RoboDK station: robot_arm.rdk

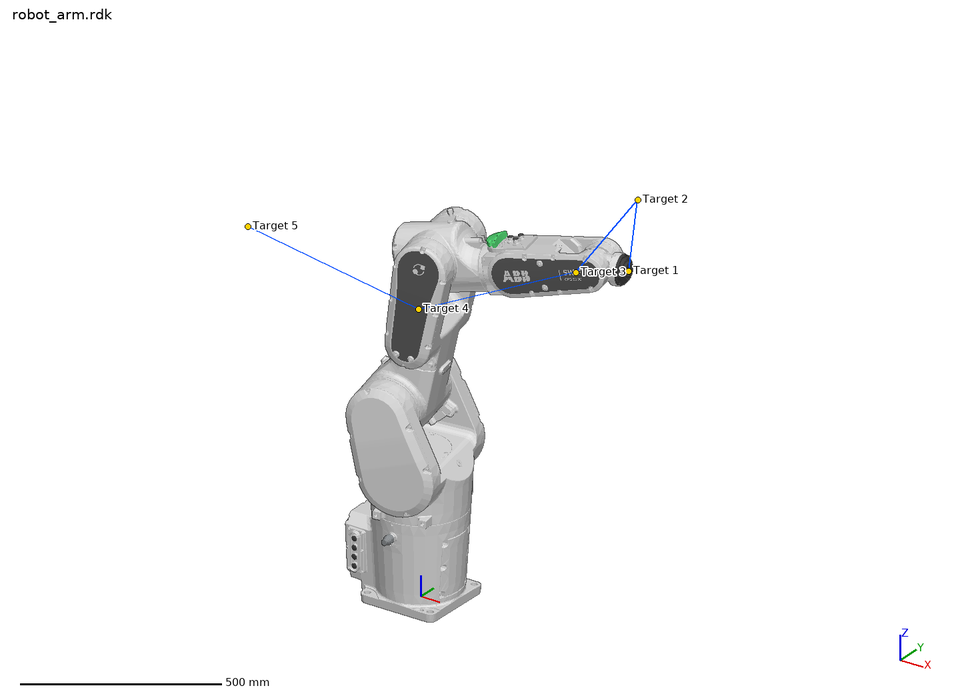
[picture v0: the station drawn from its stored meshes, robots at their saved joint values, targets as dots, program paths as lines]
Station robot_arm (saved by RoboDK 5.8.0). Poses are relative to the parent item; angles as X-Y-Z fixed-axis rotations.
  - frame ABB CRB 1300-11/0.9 Base at (0, 1000, 0) mm
    - robot ABB CRB 1300-11/0.9: 6 axes
        modified DH rows (alpha deg, a mm, theta deg, d mm): 0, 0, 0, 544; -90, 50, -90, 0; 0, 425, 0, 0; -90, 40, 0, 425; 90, 0, 0, 0; -90, 0, 180, 90
        joint limits [-180, -100, -210, -230, -130, -242] to [180, 130, 65, 230, 130, 242]; home [0, 0, 0, 0, 0, 0]; saved at [-169.09, -13.79, -153.79, -179.99, 12.4, 0]
    - target Target 1 (Cartesian target) at (554.75, 106.93, 1009.12) mm, rotated rx 26.03 ry 89.98 rz 36.94 deg; joints [-169.09, -13.79, -153.79, -179.99, 12.4, 0] of ABB CRB 1300-11/0.9
    - target Target 2 (Cartesian target) at (342.12, 449.59, 1009.12) mm, rotated rx 26.03 ry 89.98 rz 78.76 deg; joints [-127.27, -13.79, -153.79, -179.99, 12.4, 0] of ABB CRB 1300-11/0.9
    - target Target 3 (Cartesian target) at (-34.26, 718.46, 596.2) mm, rotated rx 179.98 ry 56.8 rz -87.29 deg; joints [-87.27, -47.01, -153.79, -179.99, 12.4, 0] of ABB CRB 1300-11/0.9
    - target Target 4 (Cartesian target) at (-369.45, 518.9, 480.16) mm, rotated rx 179.98 ry 40.97 rz -54.58 deg; joints [-54.55, -47, -169.64, -179.98, 12.39, 0] of ABB CRB 1300-11/0.9
    - target Target 5 (Cartesian target) at (-573.83, 73.2, 828.79) mm, rotated rx 179.94 ry 70.66 rz -7.33 deg; joints [-7.27, -17.32, -169.63, -179.98, 12.39, 0] of ABB CRB 1300-11/0.9
  - program Prog1 (6 instructions, listed below)
  - Python program Prog2 (listed below)
  - Python program Prog3 (listed below)
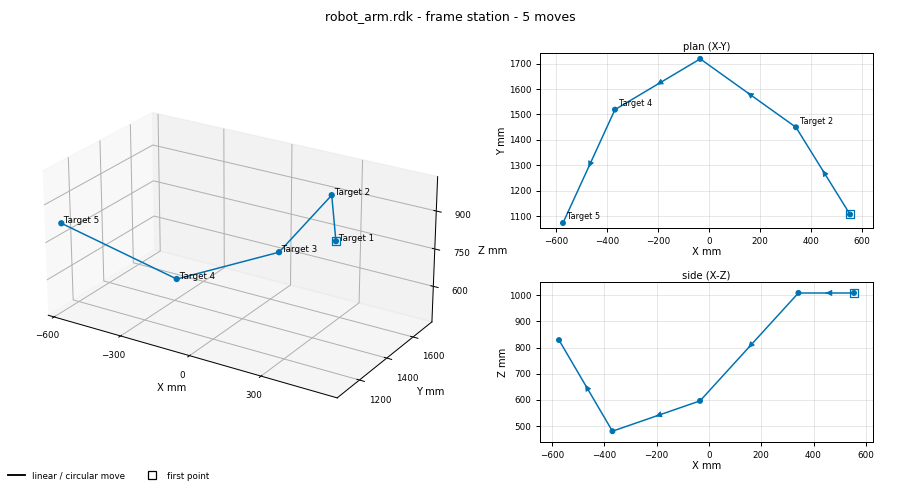
[picture p0: tool path of robot_arm.rdk in frame station, 5 of 5 moves have a stored position in this frame; points joined in program order, loops and branches not executed]

--- program Prog1 (robot ABB CRB 1300-11/0.9) ---
  Set Ref.: ABB CRB 1300-11/0.9 Base
  MoveJ (Target 1)
  MoveL (Target 2)
  MoveL (Target 3)
  MoveL (Target 4)
  MoveL (Target 5)

--- Python program Prog2 ---
# RoboDK and OpenCV hand gesture control script
from robolink import *    # RoboDK's API
from robodk import *      # Math toolbox for robots

# Starwt the RoboDK API:
RDK = Robolink()

# Get the robot (first robot found):
robot = RDK.Item('', ITEM_TYPE_ROBOT)

# Get the reference targets by name:
target = RDK.Item('Target 1')
target2 = RDK.Item('Target 2')
target3 = RDK.Item('Target 3')
target4 = RDK.Item('Target 4')
target5 = RDK.Item('Target 5')

# Move the robot to the reference point:
robot.MoveJ(target)

## Vision-based control ##
# The program moves the robot to different targets based on hand gestures (fingers raised)

import cv2 as cv
import mediapipe as mp
import time
import math

def findPos(img, results, handNumb=0, draw=False, palmLM=False, drawPalm=False):
    lmList = []
    if results.multi_hand_landmarks:
        myHand = results.multi_hand_landmarks[handNumb]
        for i, lm in enumerate(myHand.landmark):
            h, w, c = img.shape
            cx, cy, cz = int(lm.x * w), int(lm.y * h), lm.z
            lmList.append([i, cx, cy, cz])
            if draw:
                cv.circle(img, (cx, cy), 5, (255, 255, 0), cv.FILLED)
        if palmLM:
            palmMarks = [0, 1, 5, 9, 13, 17]
            palmX, palmY, palmZ = 0, 0, 0
            for id in palmMarks:
                palmX += lmList[id][1]
                palmY += lmList[id][2]
                palmZ += lmList[id][3]
            palm = [21, int(palmX / 6), int(palmY / 6), palmZ / 6]
            lmList.append(palm)
            if drawPalm:
                cv.circle(img, (palm[1], palm[2]), 5, (255, 255, 0), cv.FILLED)
    return lmList

def lmDistance(lm1, lm2):
    dx = lm2[1] - lm1[1]
    dy = lm2[2] - lm1[2]
    dist = math.sqrt((dx ** 2) + (dy ** 2))
    return int(dist)

def fingersState(lmList):
    fingersUp = []
    fingersCount = 0
    tipIds = [4, 8, 12, 16, 20]
    for id in tipIds:
        if id == 4:
            distP = lmDistance(lmList[id], lmList[17])
            distF = lmDistance(lmList[id - 2], lmList[17])
        else:
            distP = lmDistance(lmList[id], lmList[0])
            distF = lmDistance(lmList[id - 2], lmList[0])
        if distP > distF:
            fingersCount += 1
            fingersUp.append(1)
        else:
            fingersUp.append(0)
    return fingersUp, fingersCount


cap = cv.VideoCapture(0)
mpHands = mp.solutions.hands
hands = mpHands.Hands()
mpDraw = mp.solutions.drawing_utils

pTime = 0
cTime = 0

while True:
    success, frame = cap.read()
    frame = cv.flip(frame, 1)
    frameRGB = cv.cvtColor(frame, cv.COLOR_BGR2RGB)
    results = hands.process(frameRGB)
    lmList = findPos(frame, results, handNumb=0, draw=True, palmLM=False, drawPalm=False)

    if len(lmList) != 0:
        fingerState, fingersCount = fingersState(lmList)
        cv.putText(frame, 'FingerState:' + str(fingerState), (20, 100), cv.FONT_HERSHEY_COMPLEX, 0.5, (0, 255, 0), thickness=1)

        # Based on the fingers raised, move to a specific target
        if fingerState == [0, 1, 0, 0, 0]:
            cv.putText(frame, 'Target 1', (200, 300), cv.FONT_HERSHEY_COMPLEX, 1, (0, 0, 255), thickness=1)
            robot.MoveJ(target)
        elif fingerState == [0, 1, 1, 0, 0]:
            cv.putText(frame, 'Target 2', (200, 300), cv.FONT_HERSHEY_COMPLEX, 1, (0, 0, 255), thickness=1)
            robot.MoveJ(target2)
        elif fingerState == [0, 1, 1, 1, 0]:
            cv.putText(frame, 'Target 3', (200, 300), cv.FONT_HERSHEY_COMPLEX, 1, (0, 0, 255), thickness=1)
            robot.MoveJ(target3)
        elif fingerState == [0, 1, 1, 1, 1]:
            cv.putText(frame, 'Target 4', (200, 300), cv.FONT_HERSHEY_COMPLEX, 1, (0, 0, 255), thickness=1)
            robot.MoveJ(target4)
        elif fingerState == [1, 1, 1, 1, 1]:
            cv.putText(frame, 'Target 5', (200, 300), cv.FONT_HERSHEY_COMPLEX, 1, (0, 0, 255), thickness=1)
            robot.MoveJ(target5)
        robot.RunInstruction('Program_Done')

    cTime = time.time()
    fps = 1 / (cTime - pTime)
    pTime = cTime

    cv.putText(frame, 'FPS: ' + str(int(fps)), (20, 40), cv.FONT_HERSHEY_COMPLEX, 1, (0, 255, 0), thickness=2)

    cv.imshow('Video', frame)
    if cv.waitKey(20) & 0xFF == 27:
        break

cap.release()
cv.destroyAllWindows()

# Trigger a program call at the end of the movement
robot.RunInstruction('Program_Done')

--- Python program Prog3 ---
# Type help("robodk.robolink") or help("robodk.robomath") for more information
# Press F5 to run the script
# Documentation: https://robodk.com/doc/en/RoboDK-API.html
# Reference:     https://robodk.com/doc/en/PythonAPI/robodk.html
# Note: It is not required to keep a copy of this file, your Python script is saved with your RDK project

# You can also use the new version of the API:
from robodk import robolink    # RoboDK API
from robodk import robomath    # Robot toolbox
import cv2
RDK = robolink.Robolink()

# Forward and backwards compatible use of the RoboDK API:
# Remove these 2 lines to follow python programming guidelines
from robodk import *      # RoboDK API
from robolink import *    # Robot toolbox
# Link to RoboDK
# RDK = Robolink()

# Notify user:
print('To edit this program:\nright click on the Python program, then, select "Edit Python script"')

# Program example:
item = RDK.Item('base')
if item.Valid():
    print('Item selected: ' + item.Name())
    print('Item posistion: ' + repr(item.Pose()))

print('Items in the station:')
itemlist = RDK.ItemList()
print(itemlist)


cap = cv2.VideoCapture(0)

if not cap.isOpened():
    print("Camera could not be opened!")
    exit()

while True:
    ret, frame = cap.read()
    if not ret:
        print("Failed to grab frame")
        break
    cv2.imshow('Test', frame)

    if cv2.waitKey(1) == 27:  # Press 'ESC' to exit
        break

cap.release()
cv2.destroyAllWindows()
# Provoking an exception will display the console output if you run this script from RoboDK
raise Exception('Program not edited.')
